FUNCTION_BLOCK MAKE_BOOL_ARRAY (* Make a new Bool Array *)
  (* Description: This program and the accompanying materials are made available under the terms of the Eclipse Public License 2.0 which is available at https://www.eclipse.org/legal/epl-2.0/ SPDX-License-Identifier: EPL-2.0 *)
  (* Version 1.0, 2026-01-02, Unknown, Unknown *)
  PACKAGE isobus::pgn::transport;
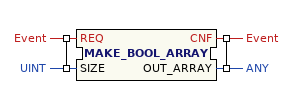
  EVENT_INPUT
    REQ WITH SIZE; (* Service Request *)
  END_EVENT
  EVENT_OUTPUT
    CNF WITH OUT_ARRAY; (* Confirmation of Requested Service *)
  END_EVENT
  VAR_INPUT
    SIZE : UINT; (* size *)
  END_VAR
  VAR_OUTPUT
    OUT_ARRAY : ANY; (* resulting array after set *)
  END_VAR
END_FUNCTION_BLOCK
